# EPICS autosave request: iocBoot/ioc13idd_dante1/auto_settings.req
file "dante_settings.req",        P=$(P), R=$(R)
file "danteN_settings.req",       P=$(P), R=$(R)
file "mca_settings.req",          P=$(P), M=$(M)
file "commonPlugin_settings.req", P=$(P)
